Staubli VAL3: OnF4.pgx

program OnF4()
begin
end
